% RSLogix 500 project btc_sin.RSS, saved by version 8.30.00.16 %
PROJECT "ML1100"    % processor: Bul.1763 MicroLogix 1100 Series A; MAIN_PROG %

PROGRAM FILES
  LAD 2 "MAIN_PROG"  7 rungs
  LAD 228 "OUTER_SIN"  10 rungs  % Constrained Sine Outer Subr:  constrain arg %
  LAD 238 "INNER_SIN"  3 rungs  % Constrained Sine Inner Subr:  Cheby approx %
  LAD 248 "INNER_COS"  3 rungs

DATA FILES
  O0 OUTPUT  4 elements
  I1 INPUT  6 elements
  S2 STATUS  66 elements
  B3 BINARY  20 elements
  T4 TIMER  10 elements
  C5 COUNTER  10 elements
  R6 CONTROL  10 elements
  N7 INTEGER  100 elements
  F8 FLOAT  181 elements
  F100 X_RADIANS  181 elements
  F101 SIN(X)  181 elements
  B223   2 elements
  N226 INTS 228  1 elements
  F227 FLOATS 228  11 elements  % Floats for LAD 228 %
  B228 CMTBITS228  16 elements
  F237 FLOATS 238  11 elements  % Floats for inner sine approximation %
  F247 FLOATS 248  11 elements  % Floats for inner cosine approximation %

LADDER 2 "MAIN_PROG"
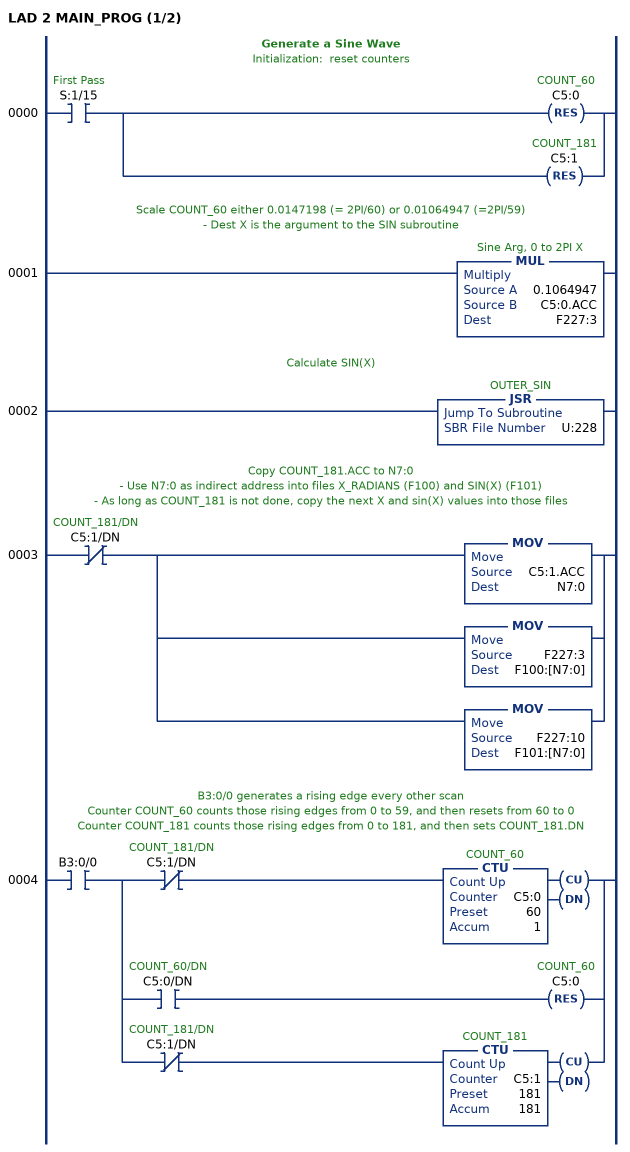
% Rung: 0 %
% TITLE: Generate a Sine Wave %
% Initialization:  reset counters %
SOR XIC S:1/15 BST RES C5:0 NXB RES C5:1 BND EOR
%   S:1/15  "First Pass" %
%   C5:0  COUNT_60 %
%   C5:1  COUNT_181 %
% Rung: 1 %
% Scale COUNT_60 either 0.0147198 (= 2PI/60) or 0.01064947 (=2PI/59)
% - Dest X is the argument to the SIN subroutine %
SOR MUL 0.1064947 C5:0.ACC F227:3 EOR
%   C5:0  COUNT_60 %
%   F227:3  X  "Sine Arg, 0 to 2PI" %
% Rung: 2 %
% Calculate SIN(X) %
SOR JSR U:228 EOR
%   U:228  OUTER_SIN %
% Rung: 3 %
% Copy COUNT_181.ACC to N7:0
% - Use N7:0 as indirect address into files X_RADIANS (F100) and SIN(X) (F101)
% - As long as COUNT_181 is not done, copy the next X and sin(X) values into those files %
SOR XIO C5:1/DN BST MOV C5:1.ACC N7:0 NXB MOV F227:3 F100:[N7:0] NXB MOV F227:10 F101:[N7:0] BND EOR
%   C5:1  COUNT_181 %
%   F227:3  X  "Sine Arg, 0 to 2PI" %
%   F227:10  SIN_RESULT  "SINE approx result" %
% Rung: 4 %
% B3:0/0 generates a rising edge every other scan
% Counter COUNT_60 counts those rising edges from 0 to 59, and then resets from 60 to 0
% Counter COUNT_181 counts those rising edges from 0 to 181, and then sets COUNT_181.DN %
SOR XIC B3:0/0 BST XIO C5:1/DN CTU C5:0 60 1 NXB XIC C5:0/DN RES C5:0 NXB XIO C5:1/DN CTU C5:1 181 181 BND EOR
%   C5:1  COUNT_181 %
%   C5:0  COUNT_60 %

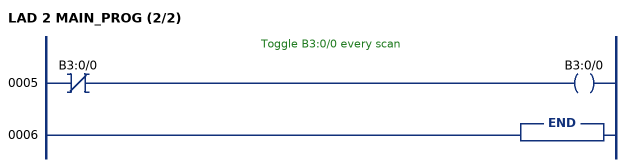
% Rung: 5 %
% Toggle B3:0/0 every scan %
SOR XIO B3:0/0 OTE B3:0/0 EOR
% Rung: 6 %
SOR END EOR

LADDER 228 "OUTER_SIN"    % Constrained Sine Outer Subr:  constrain arg %
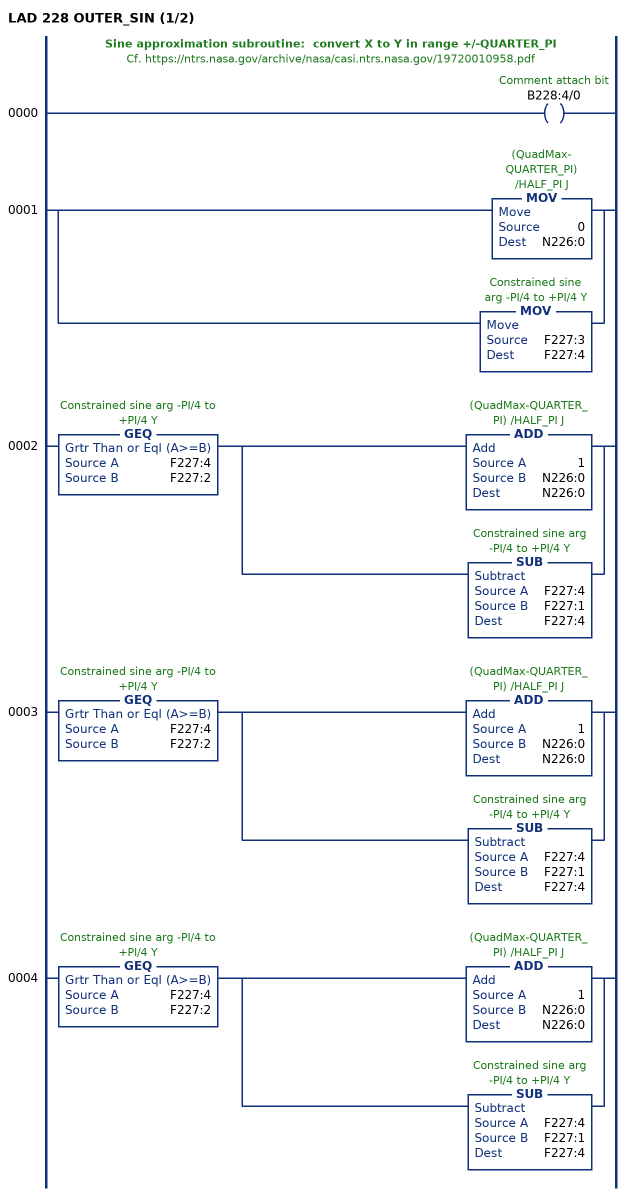
% Rung: 0 %
% TITLE: Sine approximation subroutine:  convert X to Y in range +/-QUARTER_PI %
% Cf. https://ntrs.nasa.gov/archive/nasa/casi.ntrs.nasa.gov/19720010958.pdf %
SOR OTE B228:4/0 EOR
%   B228:4/0  "Comment attach bit" %
% Rung: 1 %
SOR BST MOV 0 N226:0 NXB MOV F227:3 F227:4 BND EOR
%   N226:0  J  "(QuadMax-QUARTER_PI) /HALF_PI" %
%   F227:3  X  "Sine Arg, 0 to 2PI" %
%   F227:4  Y  "Constrained sine arg -PI/4 to +PI/4" %
% Rung: 2 %
SOR GEQ F227:4 F227:2 BST ADD 1 N226:0 N226:0 NXB SUB F227:4 F227:1 F227:4 BND EOR
%   F227:4  Y  "Constrained sine arg -PI/4 to +PI/4" %
%   F227:2  QUARTER_PI %
%   N226:0  J  "(QuadMax-QUARTER_PI) /HALF_PI" %
%   F227:1  HALF_PI %
% Rung: 3 %
SOR GEQ F227:4 F227:2 BST ADD 1 N226:0 N226:0 NXB SUB F227:4 F227:1 F227:4 BND EOR
%   F227:4  Y  "Constrained sine arg -PI/4 to +PI/4" %
%   F227:2  QUARTER_PI %
%   N226:0  J  "(QuadMax-QUARTER_PI) /HALF_PI" %
%   F227:1  HALF_PI %
% Rung: 4 %
SOR GEQ F227:4 F227:2 BST ADD 1 N226:0 N226:0 NXB SUB F227:4 F227:1 F227:4 BND EOR
%   F227:4  Y  "Constrained sine arg -PI/4 to +PI/4" %
%   F227:2  QUARTER_PI %
%   N226:0  J  "(QuadMax-QUARTER_PI) /HALF_PI" %
%   F227:1  HALF_PI %

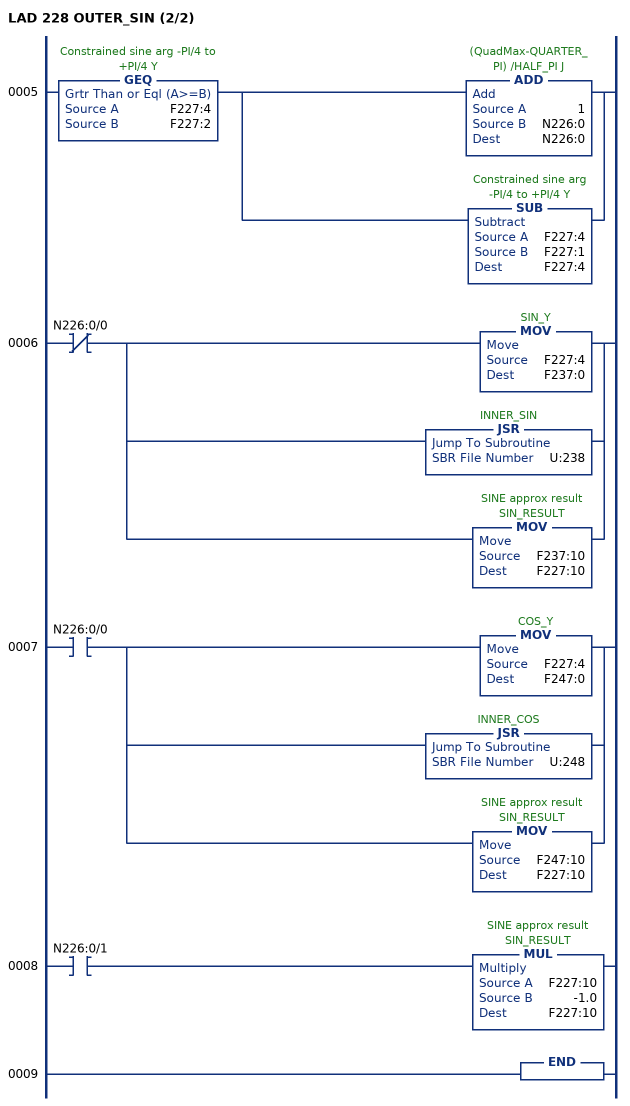
% Rung: 5 %
SOR GEQ F227:4 F227:2 BST ADD 1 N226:0 N226:0 NXB SUB F227:4 F227:1 F227:4 BND EOR
%   F227:4  Y  "Constrained sine arg -PI/4 to +PI/4" %
%   F227:2  QUARTER_PI %
%   N226:0  J  "(QuadMax-QUARTER_PI) /HALF_PI" %
%   F227:1  HALF_PI %
% Rung: 6 %
SOR XIO N226:0/0 BST MOV F227:4 F237:0 NXB JSR U:238 NXB MOV F237:10 F227:10 BND EOR
%   F227:4  Y  "Constrained sine arg -PI/4 to +PI/4" %
%   F237:0  SIN_Y %
%   U:238  INNER_SIN %
%   F237:10  INNER_SIN_RESULT %
%   F227:10  SIN_RESULT  "SINE approx result" %
% Rung: 7 %
SOR XIC N226:0/0 BST MOV F227:4 F247:0 NXB JSR U:248 NXB MOV F247:10 F227:10 BND EOR
%   F227:4  Y  "Constrained sine arg -PI/4 to +PI/4" %
%   F247:0  COS_Y %
%   U:248  INNER_COS %
%   F247:10  INNER_COS_RESULT %
%   F227:10  SIN_RESULT  "SINE approx result" %
% Rung: 8 %
SOR XIC N226:0/1 MUL F227:10 -1.0 F227:10 EOR
%   F227:10  SIN_RESULT  "SINE approx result" %
% Rung: 9 %
SOR END EOR

LADDER 238 "INNER_SIN"    % Constrained Sine Inner Subr:  Cheby approx %
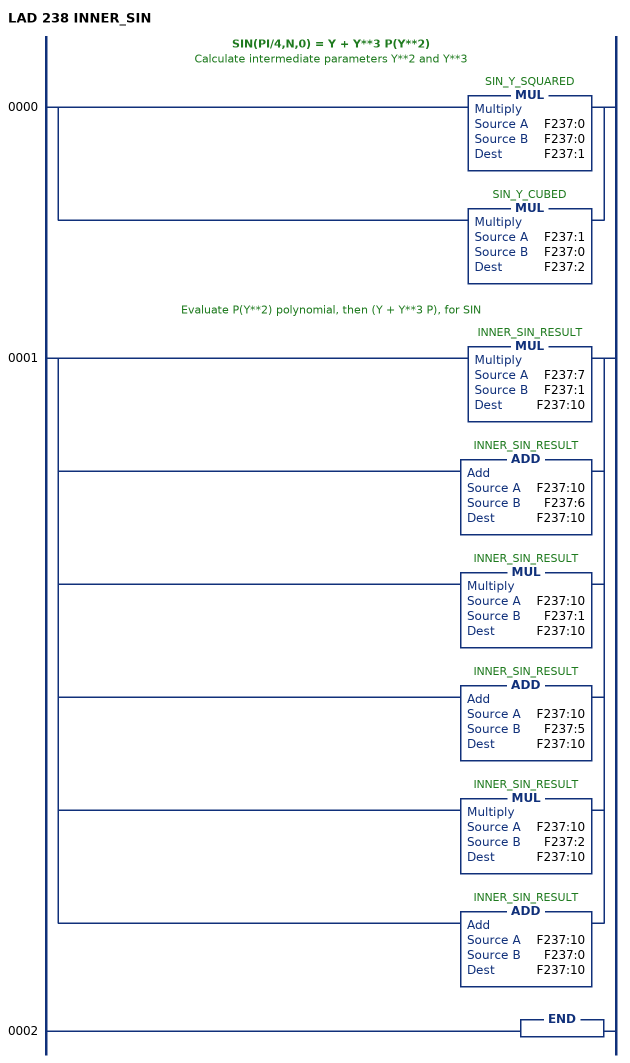
% Rung: 0 %
% TITLE: SIN(PI/4,N,0) = Y + Y**3 P(Y**2) %
% Calculate intermediate parameters Y**2 and Y**3 %
SOR BST MUL F237:0 F237:0 F237:1 NXB MUL F237:1 F237:0 F237:2 BND EOR
%   F237:0  SIN_Y %
%   F237:1  SIN_Y_SQUARED %
%   F237:2  SIN_Y_CUBED %
% Rung: 1 %
% Evaluate P(Y**2) polynomial, then (Y + Y**3 P), for SIN %
SOR BST MUL F237:7 F237:1 F237:10 NXB ADD F237:10 F237:6 F237:10 NXB MUL F237:10 F237:1 F237:10 NXB ADD F237:10 F237:5 F237:10 NXB MUL F237:10 F237:2 F237:10 NXB ADD F237:10 F237:0 F237:10 BND EOR
%   F237:7  SIN_P02 %
%   F237:1  SIN_Y_SQUARED %
%   F237:10  INNER_SIN_RESULT %
%   F237:6  SIN_P01 %
%   F237:5  SIN_P00 %
%   F237:2  SIN_Y_CUBED %
%   F237:0  SIN_Y %
% Rung: 2 %
SOR END EOR

LADDER 248 "INNER_COS"
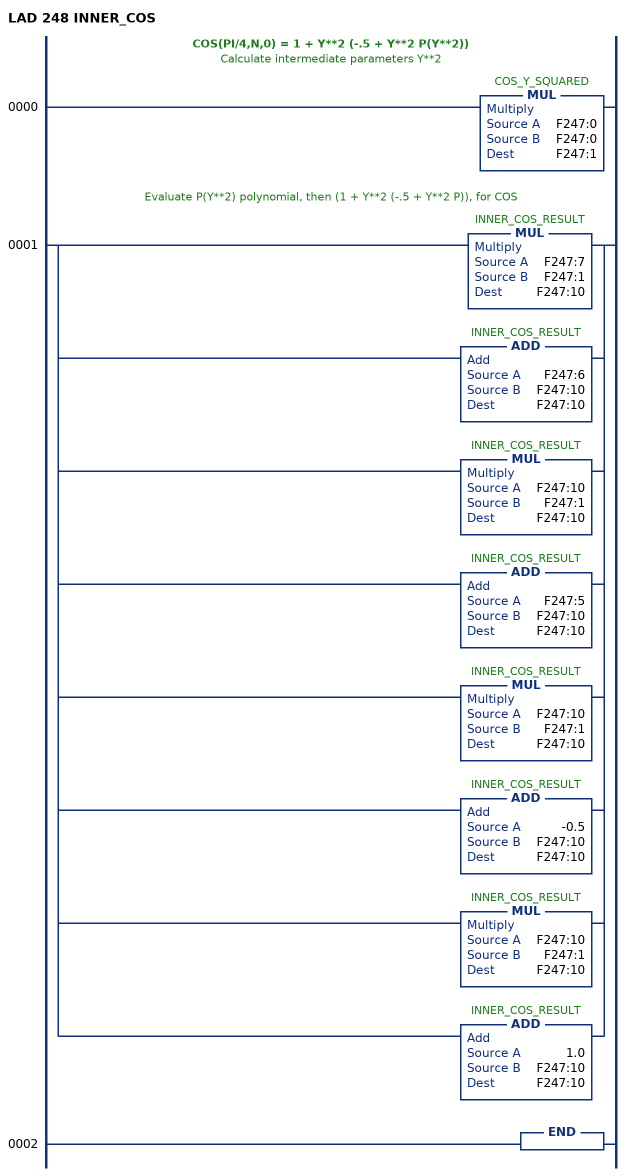
% Rung: 0 %
% TITLE: COS(PI/4,N,0) = 1 + Y**2 (-.5 + Y**2 P(Y**2)) %
% Calculate intermediate parameters Y**2 %
SOR MUL F247:0 F247:0 F247:1 EOR
%   F247:0  COS_Y %
%   F247:1  COS_Y_SQUARED %
% Rung: 1 %
% Evaluate P(Y**2) polynomial, then (1 + Y**2 (-.5 + Y**2 P)), for COS %
SOR BST MUL F247:7 F247:1 F247:10 NXB ADD F247:6 F247:10 F247:10 NXB MUL F247:10 F247:1 F247:10 NXB ADD F247:5 F247:10 F247:10 NXB MUL F247:10 F247:1 F247:10 NXB ADD -0.5 F247:10 F247:10 NXB MUL F247:10 F247:1 F247:10 NXB ADD 1.0 F247:10 F247:10 BND EOR
%   F247:7  COS_P02 %
%   F247:1  COS_Y_SQUARED %
%   F247:10  INNER_COS_RESULT %
%   F247:6  COS_P01 %
%   F247:5  COS_P00 %
% Rung: 2 %
SOR END EOR

OTHER DOCUMENTED ADDRESSES
  B228:4/1  "Comment attach bit"
  DFILE:0  "OUTPUT"
  DFILE:1  "INPUT"
  DFILE:2  "STATUS"
  DFILE:3  "BINARY"
  DFILE:4  "TIMER"
  DFILE:5  "COUNTER"
  DFILE:6  "CONTROL"
  DFILE:7  "INTEGER"
  DFILE:8  "FLOAT"
  DFILE:10  "PID_PARAM"
  DFILE:13  "PID_STATUS"
  DFILE:17  "PID_CS PID Control Loop Com mand & Status Data"
  DFILE:18  "PID_LOOP Individual PID Contr ol Loop Data File"
  DFILE:77  "PID_CW A PID Control Loop Sub routine Cmd & Status Data File"
  DFILE:88  "PID_DATA_A PID Control Loop Sub routine Master Data File"
  DFILE:200  "Split Range Time Pro portioned Data file"
  DFILE:233  "SR_TP_BIN Split Range Time Pro portioned Reall Data File"
  DFILE:234  "SR_TP_TMR Split Range Time Pro portioned Timer Data File"
  DFILE:237  "SR_TP_INT Split Range Time Pro portioned Integer Da ta File"
  DFILE:238  "SR_TP_REAL Split Range Time Pro portioned Reall Data File"
  DFILE:247  "PID_CW PID Control Loop Sub routine Cmd & Status Data File"
  DFILE:248  "PID_DATA PID Control Loop Sub routine Master Data File"
  DFILE:253  "PID_BINARY PID"
  F227:0  TWO_PI
  PFILE:3  "Motor Starter Contro l Subroutine"
  PFILE:4  "PID Control Loop Sub routine"
  PFILE:5  "Deadtime Delay Subro utine"
  PFILE:228  "Deadtime Delay Progr am File"
  PFILE:238  "Constrained Sine sub routine:  Constraine dChebyshev"
  PFILE:248  "Multiple PID Floatin g Point Subroutine"

COMMENTS NOT ATTACHED TO A CURRENT RUNG
  B3:9/2: Motor #3 External Toggle Pushbutton Controlled Start /. Stop Logic with One Shot Functionality & No One Shot Instructions
  B3:9/1: Motor #2 HMI Interface Toggle Pushbutton Start /. Stop Logic - One Shot Instruction Not Required
  O:0.0/0: Motor Starter Programming Example / ******
    Motor #1 HMI Interface Start /. Stop & Run Time Logic
    ******
  B3:6/0: ******
    Pilot Light "Flasher Bit" Logic: ON for 1.0 Seconds and OFF for 2.0 Seconds with ONE (1) Timer !!! (pjc - 02/03/2020)
    ******
  B3:9/0: MicroLogix Test Program of sine function over sixty steps
  N17:0/1: PID Control Loop #1 / ******
    Auto / Manual Mode Logic
    ******
  N17:1/1: PID Control Loop #2 / ******
    Auto / Manual Mode Logic
    ******
  B253:0/0: ******
    SP & PV Scalling & Erro Calculations
    ******
  B253:0/1: ******
    Calculate Absolute Value of Percent Errir & Percent Deadband
    ******
  B253:0/2: ******
    PID Control Loop #1 Proportinal / Integral / Derivative Calclulations IF Absolute Value of Percent Error => Percent Deadband
    ******
  B253:0/3: ******
    PID Control Loop #1 Calculate Total Auto Mode Output = P Term + I Term + D Term
    ******
  B253:0/4: ******
    PID Control Loop #1 Auto Mode Anti-Reset Windup if Total Auto Output is Less Than 0.0%
    ******
  B253:0/5: ******
    PID Control Loop #1 Auto Mode Anti-Reset Windup if Total Auto Output is Greater Than 100.0%
    ******
  B233:0/4: ******
    If F238:0 Input < 0.0% Then Calculate Cooling On & Off Timer Presets
    ******
  B233:0/3: ******
    Heat Timer On / Off and Heat Output Logic
    ******
  B233:0/2: ******
    If F238:0 Input > 0.0% Then Calculate Heating On & Off Timer Presets
    ******
  B233:0/1: Split Range Time Proportioning Subroutine / ******
    Check that the Split Range Input (F238:0) & Maximum Heating Limit (F238:1) & the Minimum Cooling Limit (F238:2) are not out of range (> 100.0% and < -100.0%)
    ******
  B233:0/0: Split Range Time Proportioning Subroutine / ******
    Calculate Heating & Cooling Scale Factors and Total Counts for Heating & Cooling Timers
    ******
  B253:0/6: ******
    PID Control Loop #1 Auto to Manual Mode Balanceles Bumpless Transfer Logic
    ******
  B253:0/7: ******
    PID Control Loop #1 Integral Term Calculation for Manual to Auto Mode Balanceles Bumpless Transfer
    ******
  B3:9/3: ******
    PID Control Loop Timing & Index Counter Logic
    ******
  B3:10/0: ******
    PID Control Loop #1 Suborutine Jump Logic
    ******
  B3:10/1: ******
    Scale & Send PID Control Loop Output to Split Range Time Proportioning Subroutine and Calculate the next PV from PID Control Loop #1 Output
    ******
  B3:10/2: ******
    PID Control Loop #2 Suborutine Jump Logic
    ******
  B3:10/3: ******
    Calculate the next PID #2 PV from PID Control Loop #1 Output
    ******
  B233:0/5: ******
    Cooling Timer On / Off and Heat Output Logic
    ******
  B243:0/1: ******
    Calculate Absolute Value of Percent Errir & Percent Deadband
    ******
  B243:0/0: PID Control Subroutine / ******
    SP & PV Scalling & Erro Calculations
    ******
  B243:0/7: ******
    PID Control Loop #1 Integral Term Calculation for Manual to Auto Mode Balanceles Bumpless Transfer
    ******
  B243:0/6: ******
    PID Control Loop #1 Auto to Manual Mode Balanceles Bumpless Transfer Logic
    ******
  B243:0/5: ******
    PID Control Loop #1 Auto Mode Anti-Reset Windup if Total Auto Output is Greater Than 100.0%
    ******
  B243:0/4: ******
    PID Control Loop #1 Auto Mode Anti-Reset Windup if Total Auto Output is Less Than 0.0%
    ******
  B243:0/3: ******
    PID Control Loop #1 Calculate Total Auto Mode Output = P Term + I Term + D Term
    ******
  B243:0/2: ******
    PID Control Loop #1 Proportinal / Integral / Derivative Calclulations IF Absolute Value of Percent Error => Percent Deadband
    ******
  B223:4/0: Sine approximation using Chebyshev coefficient over constrained range (+/-PI/4) / Cf. https://ntrs.nasa.gov/archive/nasa/casi.ntrs.nasa.gov/19720010958.pdf
  B223:4/1: Initialization
  B223:4/2: ******
    Deadtime Logxc Counter Programming
    ******
  B223:4/3: ******
    Deadtime Logic Timer & Output Programming
    ******
  B223:4/4: ******
    Deadtime Delay Logic HMI Timer #1 Preset Count Up / Down Logic
    ******
  B228:4/1: Initialization
  U:228: Calculate SIN(X)

DATA TABLE (non-zero values as saved)
DATA B3
% B3:0 % 0X0000 0X0000 0X0000 0X0000 0X0000 0X0000 0X0001 0X0000 0X0000 0X4201
% B3:10 % 0X400A 0X0000 0X0000 0X0000 0X0000 0X0000 0X0000 0X0000 0X0000 0X0000
DATA T4
% .PRE .ACC %
% T4:0 % 1000 757
% T4:1 % 50 30
% T4:2 % 300 86
DATA C5
% .PRE .ACC %
% C5:0 % 60 1
% C5:1 % 181 181
DATA N7
% N7:0 % 180 0 0 0 0 0 0 0 0 0
% N7:10 % 100 200 0 0 0 0 0 0 0 0
DATA F100
% F100:0 % 0 0.1064947 0.2129894 0.3194841 0.4259788
% F100:5 % 0.5324735 0.6389682 0.7454629 0.8519576 0.9584523
% F100:10 % 1.064947 1.171442 1.277936 1.384431 1.490926
% F100:15 % 1.597421 1.703915 1.81041 1.916905 2.023399
% F100:20 % 2.129894 2.236389 2.342883 2.449378 2.555873
% F100:25 % 2.662368 2.768862 2.875357 2.981852 3.088346
% F100:30 % 3.194841 3.301336 3.40783 3.514325 3.62082
% F100:35 % 3.727314 3.833809 3.940304 4.046799 4.153294
% F100:40 % 4.259788 4.366283 4.472777 4.579272 4.685767
% F100:45 % 4.792262 4.898757 5.005251 5.111746 5.21824
% F100:50 % 5.324735 5.43123 5.537724 5.644219 5.750714
% F100:55 % 5.857209 5.963703 6.070198 6.176693 6.283187
% F100:60 % 0 0.1064947 0.2129894 0.3194841 0.4259788
% F100:65 % 0.5324735 0.6389682 0.7454629 0.8519576 0.9584523
% F100:70 % 1.064947 1.171442 1.277936 1.384431 1.490926
% F100:75 % 1.597421 1.703915 1.81041 1.916905 2.023399
% F100:80 % 2.129894 2.236389 2.342883 2.449378 2.555873
% F100:85 % 2.662368 2.768862 2.875357 2.981852 3.088346
% F100:90 % 3.194841 3.301336 3.40783 3.514325 3.62082
% F100:95 % 3.727314 3.833809 3.940304 4.046799 4.153294
% F100:100 % 4.259788 4.366283 4.472777 4.579272 4.685767
% F100:105 % 4.792262 4.898757 5.005251 5.111746 5.21824
% F100:110 % 5.324735 5.43123 5.537724 5.644219 5.750714
% F100:115 % 5.857209 5.963703 6.070198 6.176693 6.283187
% F100:120 % 0 0.1064947 0.2129894 0.3194841 0.4259788
% F100:125 % 0.5324735 0.6389682 0.7454629 0.8519576 0.9584523
% F100:130 % 1.064947 1.171442 1.277936 1.384431 1.490926
% F100:135 % 1.597421 1.703915 1.81041 1.916905 2.023399
% F100:140 % 2.129894 2.236389 2.342883 2.449378 2.555873
% F100:145 % 2.662368 2.768862 2.875357 2.981852 3.088346
% F100:150 % 3.194841 3.301336 3.40783 3.514325 3.62082
% F100:155 % 3.727314 3.833809 3.940304 4.046799 4.153294
% F100:160 % 4.259788 4.366283 4.472777 4.579272 4.685767
% F100:165 % 4.792262 4.898757 5.005251 5.111746 5.21824
% F100:170 % 5.324735 5.43123 5.537724 5.644219 5.750714
% F100:175 % 5.857209 5.963703 6.070198 6.176693 6.283187
DATA F101
% F101:0 % 0 0.1062935 0.2113827 0.3140768 0.4132123
% F101:5 % 0.5076659 0.5963675 0.678312 0.752571 0.818303
% F101:10 % 0.8747633 0.9213122 0.9574222 0.9826843 0.996812
% F101:15 % 0.9996456 0.9911528 0.9714298 0.9407 0.8993118
% F101:20 % 0.847734 0.7865511 0.7164562 0.6382434 0.5527992
% F101:25 % 0.4610915 0.3641596 0.2631015 0.1590624 0.05322086
% F101:30 % -0.05322348 -0.1590648 -0.2631038 -0.3641618 -0.4610937
% F101:35 % -0.5528011 -0.6382453 -0.7164578 -0.7865525 -0.8477354
% F101:40 % -0.8993129 -0.9407009 -0.9714303 -0.9911531 -0.9996457
% F101:45 % -0.9968119 -0.9826837 -0.9574215 -0.9213111 -0.8747622
% F101:50 % -0.8183016 -0.7525696 -0.6783103 -0.5963653 -0.5076641
% F101:55 % -0.4132102 -0.3140745 -0.2113801 -0.1062906 2.145767e-06
% F101:60 % 0 0.1062935 0.2113827 0.3140768 0.4132123
% F101:65 % 0.5076659 0.5963675 0.678312 0.752571 0.818303
% F101:70 % 0.8747633 0.9213122 0.9574222 0.9826843 0.996812
% F101:75 % 0.9996456 0.9911528 0.9714298 0.9407 0.8993118
% F101:80 % 0.847734 0.7865511 0.7164562 0.6382434 0.5527992
% F101:85 % 0.4610915 0.3641596 0.2631015 0.1590624 0.05322086
% F101:90 % -0.05322348 -0.1590648 -0.2631038 -0.3641618 -0.4610937
% F101:95 % -0.5528011 -0.6382453 -0.7164578 -0.7865525 -0.8477354
% F101:100 % -0.8993129 -0.9407009 -0.9714303 -0.9911531 -0.9996457
% F101:105 % -0.9968119 -0.9826837 -0.9574215 -0.9213111 -0.8747622
% F101:110 % -0.8183016 -0.7525696 -0.6783103 -0.5963653 -0.5076641
% F101:115 % -0.4132102 -0.3140745 -0.2113801 -0.1062906 2.145767e-06
% F101:120 % 0 0.1062935 0.2113827 0.3140768 0.4132123
% F101:125 % 0.5076659 0.5963675 0.678312 0.752571 0.818303
% F101:130 % 0.8747633 0.9213122 0.9574222 0.9826843 0.996812
% F101:135 % 0.9996456 0.9911528 0.9714298 0.9407 0.8993118
% F101:140 % 0.847734 0.7865511 0.7164562 0.6382434 0.5527992
% F101:145 % 0.4610915 0.3641596 0.2631015 0.1590624 0.05322086
% F101:150 % -0.05322348 -0.1590648 -0.2631038 -0.3641618 -0.4610937
% F101:155 % -0.5528011 -0.6382453 -0.7164578 -0.7865525 -0.8477354
% F101:160 % -0.8993129 -0.9407009 -0.9714303 -0.9911531 -0.9996457
% F101:165 % -0.9968119 -0.9826837 -0.9574215 -0.9213111 -0.8747622
% F101:170 % -0.8183016 -0.7525696 -0.6783103 -0.5963653 -0.5076641
% F101:175 % -0.4132102 -0.3140745 -0.2113801 -0.1062906 2.145767e-06
DATA F227
% F227:0 % 6.283185 1.570796 0.7853982 0.1064947 0.1064947
% F227:10 % 0.1062935
DATA B228
% B228:0 % 0X0000 0X0000 0X0000 0X0000 0X0001 0X0000 0X0000 0X0000 0X0000 0X0000
DATA F237
% F237:0 % 0.1064947 0.01134112 0.001207769 0 0
% F237:5 % -0.1666665 0.008332064 -0.000195022 0 0
% F237:10 % 0.1062935
DATA F247
% F247:0 % 0.7188408 0.5167322 0 0 0
% F247:5 % 0.04166664 -0.001388723 2.44231e-05 0 0
% F247:10 % 0.7525696
